// TIA Portal V20 export
ORGANIZATION_BLOCK "Startup"   // OB1005, LAD, Startup
TITLE = "Complete Restart"
AUTHOR : ERsystem_FA2_DH. Kim
// stored: AutoNumber false, IsIECCheckEnabled true, Namespace Unit1.Em0, SetENOAutomatically false
   VAR_INPUT
      LostRetentive : Bool;   // True if retentive data are lost
      LostRTC : Bool;   // True if date and time are lost
   END_VAR
BEGIN

REGION Network 1 (SCL): Build the Absolut Reference Designator
   // Set the Absoult Reference Designator in the Config DB
   IF LEN(IN := "Unit1.Em0.Config".em.referenceDesignator.parent) <> 0 THEN
     "Unit1.Em0.Config".em.referenceDesignator.combined := CONCAT_WSTRING(IN1 := "Unit1.Em0.Config".em.referenceDesignator.parent, IN2 := WSTRING#'.', IN3 := "Unit1.Em0.Config".em.referenceDesignator.relative);
   ELSE
     "Unit1.Em0.Config".em.referenceDesignator.combined := "Unit1.Em0.Config".em.referenceDesignator.relative;
   END_IF;
END_REGION

REGION Network 2 (SCL): Assign axes data
   //Assign axes
   "Unit1.Em0.Config".axis[1] := "BA030AZSDR1_UnwinderTopAxisB";

   // Assign configuration data of axis

   // Axis 1 BA030AZSDR1_UnwinderTopAxisB
   "Unit1.Em0.HmiInterface".cmUnwinderTopAxisB.commandConfiguration.jog.velocity := 10.0;
   "Unit1.Em0.HmiInterface".cmUnwinderTopAxisB.commandConfiguration.jog.acceleration := 100.0;
   "Unit1.Em0.HmiInterface".cmUnwinderTopAxisB.commandConfiguration.jog.deceleration := 100.0;
   "Unit1.Em0.HmiInterface".cmUnwinderTopAxisB.commandConfiguration.moveVelocity.velocity := 10.0;
   "Unit1.Em0.HmiInterface".cmUnwinderTopAxisB.commandConfiguration.moveVelocity.acceleration := 100.0;
   "Unit1.Em0.HmiInterface".cmUnwinderTopAxisB.commandConfiguration.moveVelocity.deceleration := 100.0;
   "Unit1.Em0.HmiInterface".cmUnwinderTopAxisB.commandConfiguration.posRelative.velocity := 10.0;
   "Unit1.Em0.HmiInterface".cmUnwinderTopAxisB.commandConfiguration.posRelative.acceleration := 100.0;
   "Unit1.Em0.HmiInterface".cmUnwinderTopAxisB.commandConfiguration.posRelative.deceleration := 100.0;

   // FB Enable
   "Unit1.Em0.HmiInterface".cmUnwinderTopAxisB.commands.enableMasterControl := TRUE;
END_REGION

REGION Network 3 (SCL): Assign TwoWayActuator data
   //Assgin Configuration data of TwoWayActuator

   "Unit1.Em0.Config".cmAirShaftTopOnOff.disableFeedbackHomePos := TRUE;
   "Unit1.Em0.Config".cmAirShaftTopOnOff.disableFeedbackWorkPos := TRUE;
END_REGION

REGION Network 4 (SCL): Assign LconSMC Config
   REGION InPut
       "Unit1.Em0.SyncNode".WinderInput.additionalVelocity := -0.5;
       "Unit1.Em0.SyncNode".WinderInput.typeOfWinder := 2;
       "Unit1.Em0.SyncNode".WinderInput.controlMode := 0;
       "Unit1.Em0.SyncNode".WinderInput.typeOfDiameterCalc := 3;
       "Unit1.Em0.SyncNode".WinderInput.holdDiameter := FALSE;
       "Unit1.Em0.SyncNode".WinderInput.setDiameter := FALSE;
       "Unit1.Em0.SyncNode".WinderInput.CntrlSetpoint := 0.0;
       "Unit1.Em0.SyncNode".WinderInput.CntrlActual := 24.9056603773585;
       "Unit1.Em0.SyncNode".WinderInput.tCycle := 2.0;
       "Unit1.Em0.SyncNode".WinderInput.winderAxis := 263;
   END_REGION

   REGION Config

       "Unit1.Em0.SyncNode".WinderConfig.positionControlled := FALSE;
       "Unit1.Em0.SyncNode".WinderConfig.axisCtrl := TRUE;
       "Unit1.Em0.SyncNode".WinderConfig.jogVelocity := 10.0;
       "Unit1.Em0.SyncNode".WinderConfig.overrideVelocity := 0.0;
       "Unit1.Em0.SyncNode".WinderConfig.maxVelocity := 100.0;
       "Unit1.Em0.SyncNode".WinderConfig.getAxisConfigAtStart := TRUE;
       "Unit1.Em0.SyncNode".WinderConfig.noOfSamplesLineVelocity := 1;

       "Unit1.Em0.SyncNode".WinderConfig.unitConfiguration.metricUnits := TRUE;
       "Unit1.Em0.SyncNode".WinderConfig.unitConfiguration.axisVelocityUnit := 1521;
       "Unit1.Em0.SyncNode".WinderConfig.unitConfiguration.axisTorqueUnit := 1126;


   //winderDynamics
       "Unit1.Em0.SyncNode".WinderConfig.winderDynamics.stopDynamics.deceleration := 360.0;
       "Unit1.Em0.SyncNode".WinderConfig.winderDynamics.stopDynamics.jerk := 0.0;
       "Unit1.Em0.SyncNode".WinderConfig.winderDynamics.stopDynamics.abortAcceleration := TRUE;
       "Unit1.Em0.SyncNode".WinderConfig.winderDynamics.syncDynamics.acceleration := 360.0;
       "Unit1.Em0.SyncNode".WinderConfig.winderDynamics.syncDynamics.deceleration := 360.0;
       "Unit1.Em0.SyncNode".WinderConfig.winderDynamics.syncDynamics.jerk := 0.0;
       "Unit1.Em0.SyncNode".WinderConfig.winderDynamics.syncDynamics.abortAcceleration := FALSE;
       "Unit1.Em0.SyncNode".WinderConfig.winderDynamics.syncDynamics.syncToleranceFactor := 1.0;
       "Unit1.Em0.SyncNode".WinderConfig.winderDynamics.operationDynamics.acceleration := 360000.0;
       "Unit1.Em0.SyncNode".WinderConfig.winderDynamics.operationDynamics.deceleration := 360000.0;
       "Unit1.Em0.SyncNode".WinderConfig.winderDynamics.operationDynamics.jerk := 0.0;
       "Unit1.Em0.SyncNode".WinderConfig.winderDynamics.jogDynamics.acceleration := 360.0;
       "Unit1.Em0.SyncNode".WinderConfig.winderDynamics.jogDynamics.deceleration := 360.0;
       "Unit1.Em0.SyncNode".WinderConfig.winderDynamics.jogDynamics.jerk := 0.0;

   //torquePrecontrolConfig
       "Unit1.Em0.SyncNode".WinderConfig.torquePrecontrolConfig.useSetValForFrictionComp := TRUE;
       "Unit1.Em0.SyncNode".WinderConfig.torquePrecontrolConfig.frictionAdjustment := 0.0;
       "Unit1.Em0.SyncNode".WinderConfig.torquePrecontrolConfig.loadGear.numerator := 30;
       "Unit1.Em0.SyncNode".WinderConfig.torquePrecontrolConfig.loadGear.denominator := 1;
       "Unit1.Em0.SyncNode".WinderConfig.torquePrecontrolConfig.MaterialWidth := 0.035;
       "Unit1.Em0.SyncNode".WinderConfig.torquePrecontrolConfig.MaterialDensity := 2700.0;
       "Unit1.Em0.SyncNode".WinderConfig.torquePrecontrolConfig.MaterialFillFactor := 1.0;
       "Unit1.Em0.SyncNode".WinderConfig.torquePrecontrolConfig.JFixed := 0.0327900014817715;
       "Unit1.Em0.SyncNode".WinderConfig.torquePrecontrolConfig.JMandrel := 0.1;
       "Unit1.Em0.SyncNode".WinderConfig.torquePrecontrolConfig.JMotor := 0.00104;
       "Unit1.Em0.SyncNode".WinderConfig.torquePrecontrolConfig.tensionAdjustment := 0.5;
       "Unit1.Em0.SyncNode".WinderConfig.torquePrecontrolConfig.accelerationAdjustment := 0.1;
       "Unit1.Em0.SyncNode".WinderConfig.torquePrecontrolConfig.dDdTAdjustment := 0.0;
       "Unit1.Em0.SyncNode".WinderConfig.torquePrecontrolConfig.upperTorqueLimit := 0.2;
       "Unit1.Em0.SyncNode".WinderConfig.torquePrecontrolConfig.lowerTorqueLimit := -0.2;
       "Unit1.Em0.SyncNode".WinderConfig.torquePrecontrolConfig.referenceTorque := 11.55;
       "Unit1.Em0.SyncNode".WinderConfig.torquePrecontrolConfig.additiveTorque := 0.0;

       //diamConfig
       "Unit1.Em0.SyncNode".WinderConfig.diamConfig.minLineVelocity := 0.5;
       "Unit1.Em0.SyncNode".WinderConfig.diamConfig.minShaftSpeed := 0.0;
       "Unit1.Em0.SyncNode".WinderConfig.diamConfig.minDia := 0.08;
       "Unit1.Em0.SyncNode".WinderConfig.diamConfig.maxDia := 0.4;
       "Unit1.Em0.SyncNode".WinderConfig.diamConfig.webThickness := 0.0001275;
       "Unit1.Em0.SyncNode".WinderConfig.diamConfig.useLineAxisActualValues := TRUE;
       "Unit1.Em0.SyncNode".WinderConfig.diamConfig.diameterSetValue := 0.1876;
       "Unit1.Em0.SyncNode".WinderConfig.diamConfig.lineFilterTime := 20.0;
       "Unit1.Em0.SyncNode".WinderConfig.diamConfig.shaftFilterTime := 20.0;
       "Unit1.Em0.SyncNode".WinderConfig.diamConfig.measuringRevolutionCount := 4.0;
       "Unit1.Em0.SyncNode".WinderConfig.diamConfig.firstDiameterOutput := 0.5;
       "Unit1.Em0.SyncNode".WinderConfig.diamConfig.diameterOutputRate := 1.0;
       "Unit1.Em0.SyncNode".WinderConfig.diamConfig.lineModLength := 1.0;
       "Unit1.Em0.SyncNode".WinderConfig.diamConfig.shaftModLength := 360.0;
       "Unit1.Em0.SyncNode".WinderConfig.diamConfig.diameterFilterTime := 360.0;
       "Unit1.Em0.SyncNode".WinderConfig.technologyControllerConfig.x1 := 0.0;
       "Unit1.Em0.SyncNode".WinderConfig.technologyControllerConfig.Kp1 := 3.0;
       "Unit1.Em0.SyncNode".WinderConfig.technologyControllerConfig.x2 := 0.0;
       "Unit1.Em0.SyncNode".WinderConfig.technologyControllerConfig.Kp2 := 0.0;
       "Unit1.Em0.SyncNode".WinderConfig.technologyControllerConfig.KpAdaptionValue := 0.0;
       "Unit1.Em0.SyncNode".WinderConfig.technologyControllerConfig.integTime := 2000.0;
       "Unit1.Em0.SyncNode".WinderConfig.technologyControllerConfig.derivTime := 0.0;
       "Unit1.Em0.SyncNode".WinderConfig.technologyControllerConfig.derivControlMode := FALSE;
       "Unit1.Em0.SyncNode".WinderConfig.technologyControllerConfig.setNominalValue := 100.0;
       "Unit1.Em0.SyncNode".WinderConfig.technologyControllerConfig.setRampTime := 10000.0;
       "Unit1.Em0.SyncNode".WinderConfig.technologyControllerConfig.filterTime := 10.0;
       "Unit1.Em0.SyncNode".WinderConfig.technologyControllerConfig.intSetValue := 0.0;
       "Unit1.Em0.SyncNode".WinderConfig.technologyControllerConfig.setIntChannel := FALSE;
       "Unit1.Em0.SyncNode".WinderConfig.technologyControllerConfig.holdIntChannel := FALSE;
       "Unit1.Em0.SyncNode".WinderConfig.technologyControllerConfig.deadBand := 0.0;
       "Unit1.Em0.SyncNode".WinderConfig.technologyControllerConfig.outValueFactor := 1.0;
       "Unit1.Em0.SyncNode".WinderConfig.technologyControllerConfig.upperLimit := 2.0;
       "Unit1.Em0.SyncNode".WinderConfig.technologyControllerConfig.lowerLimit := -2.0;
       "Unit1.Em0.SyncNode".WinderConfig.technologyControllerConfig.limRampTime := 300.0;
       "Unit1.Em0.SyncNode".WinderConfig.technologyControllerConfig.tensionReference := 0.0;
       "Unit1.Em0.SyncNode".WinderConfig.webbreakDetectionConfig.enableDetection := FALSE;
       "Unit1.Em0.SyncNode".WinderConfig.webbreakDetectionConfig.minLineVelocity := 5.0;
       "Unit1.Em0.SyncNode".WinderConfig.webbreakDetectionConfig.upperLimitError := 0.5;
       "Unit1.Em0.SyncNode".WinderConfig.webbreakDetectionConfig.lowerLimitError := 0.5;
       "Unit1.Em0.SyncNode".WinderConfig.webbreakDetectionConfig.delayTime := T#200ms;
   END_REGION
END_REGION

REGION Network 5 (SCL): Assign EPC Config
   "Unit1.Em0.Config".cmEpcTop.hwID.EkrOut_Auto_Sp_Acp_HW_ID := 1039;
   "Unit1.Em0.Config".cmEpcTop.hwID.EkrOut_CAM_Data_HW_ID := 1040;
   "Unit1.Em0.Config".cmEpcTop.hwID.EkrOut_CLS_Data_HW_ID := 1041;
   "Unit1.Em0.Config".cmEpcTop.hwID.EkrOut_Guiding_edges_HW_ID := 1043;
   "Unit1.Em0.Config".cmEpcTop.hwID.EkrOut_HEADER_Data_HW_ID := 1044;
   "Unit1.Em0.Config".cmEpcTop.hwID.EkrOut_POS_unit_HW_ID := 1046;
   "Unit1.Em0.Config".cmEpcTop.hwID.EkrOut_SEN_Data_HW_ID := 1047;
   "Unit1.Em0.Config".cmEpcTop.hwID.EkrOut_Servo_Center_HW_ID := 1048;
   "Unit1.Em0.Config".cmEpcTop.hwID.EkrOut_Setpoint_HW_ID := 1049;
   "Unit1.Em0.Config".cmEpcTop.hwID.EkrOut_Web_width_HW_ID := 1050;
   "Unit1.Em0.Config".cmEpcTop.hwID.EkrIn_Auto_Sp_Acp_HW_ID := 1051;
   "Unit1.Em0.Config".cmEpcTop.hwID.EkrIn_HEADER_Data_HW_ID := 1053;
   "Unit1.Em0.Config".cmEpcTop.hwID.EkrIn_POS_unit_HW_ID := 1055;
   "Unit1.Em0.Config".cmEpcTop.hwID.EkrIn_Setpoint_HW_ID := 1056;
   "Unit1.Em0.Config".cmEpcTop.hwID.EkrIn_Web_width_HW_ID := 1057;
END_REGION
END_ORGANIZATION_BLOCK
